SYSTEM Test_5 (* System Configuration *)
  (* Standard: 61499-1 *)
  (* Version 0.3, 2003-12-05, JHC, Rockwell Automation, Renamed from NEWSYSTEM. *)
  (* Version 0.2, 2002-11-05, JHC, Rockwell Automation, Fixed missing (empty) FBD in Application. *)
  (* Version 0.1, 2002-01-17, JHC, Rockwell Automation, Minor cleanup *)
  (* Version 0.0, 2000-05-27, JHC, Rockwell Automation *)
  APPLICATION APP1
  END_APPLICATION
  DEVICE DEV1 : FRAME_DEVICE(BOUNDS := [110,110,110,110], GRID := [1,1])
    RESOURCE RES1 : PANEL_RESOURCE(ROWS := 1, COLS := 1)
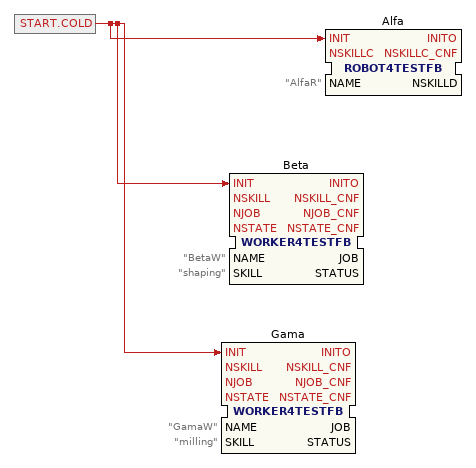
      FBS
        Alfa : ROBOT4TESTFB(NAME := "AlfaR");
        Beta : WORKER4TESTFB(SKILL := "shaping", NAME := "BetaW");
        Gama : WORKER4TESTFB(NAME := "GamaW", SKILL := "milling");
      END_FBS
      EVENT_CONNECTIONS
        START.COLD TO Alfa.INIT;
        START.COLD TO Beta.INIT;
        START.COLD TO Gama.INIT;
      END_CONNECTIONS
    END_RESOURCE
  END_DEVICE
END_SYSTEM
